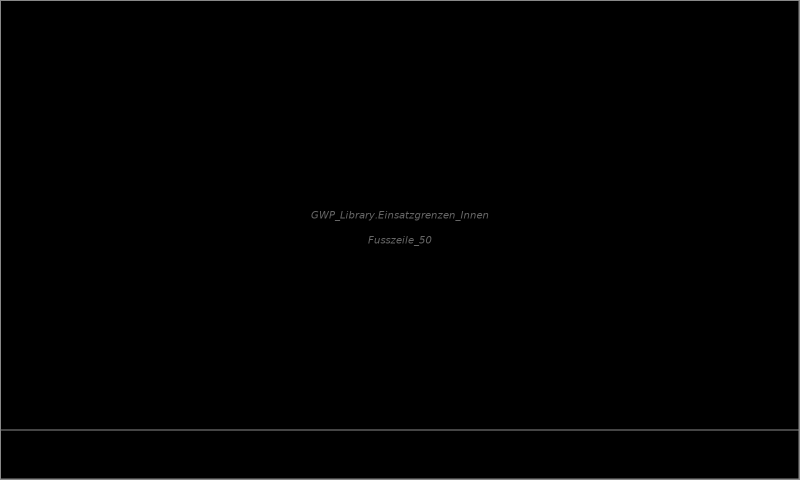
VISUALIZATION EG_Innen  // 800x480
    Frame (0,0 800x430)
        shows GWP_Library.Einsatzgrenzen_Innen(FB_Einsatzgrenzen_Innen := Main.Kreis_3KO_0.Einsatzgrenzen_Innen)
    Frame (0,0 800x480)
        shows Fusszeile_50()
END_VISUALIZATION

(* stored: Version 1.1.0.1, ProductVersion 3.1.4022.6
   Visu EG_Innen: Id {76af3358-981a-4ad5-b570-035fd80805ba} *)
